PROGRAM PRG_ManualControl
VAR
END_VAR

END_PROGRAM

(* stored: Version 1.1.0.1, ProductVersion 3.1.4024.12
   POU PRG_ManualControl: Id {d07ba183-6201-49c6-acdd-4e668144af08}, SpecialFunc None *)
